PROGRAM MAIN
VAR
END_VAR

END_PROGRAM

(* stored: Version 1.1.0.1
   POU MAIN: Id {5db1f1aa-4e41-4b0b-bbd6-6aa4de31c8c8} *)
